TYPE Replenishment_Module :
STRUCT
	infeed : ARRAY[0..1]OF Infeed;
	outfeed : ARRAY[0..1]OF Outfeed;
	lift : ARRAY[0..1]OF Lift;
END_STRUCT
END_TYPE

(* stored: Version 1.1.0.1, ProductVersion 3.1.4024.12
   DUT Replenishment_Module: Id {397c471c-4a09-425a-bc1e-d80e3a5d0a90} *)
